TYPE ST_EtherCATSlaveInfo :
STRUCT
	nAddr 			: UDINT;
	nlinkState		: UDINT;
	edeviceState	: ST_EcSlaveState;
	sType 			: STRING[16];
	sName 			: STRING[32];
END_STRUCT
END_TYPE

(* stored: Version 1.1.0.1, ProductVersion 3.1.4024.15
   DUT ST_EtherCATSlaveInfo: Id {60ac04a1-ff09-493a-a681-f256502520e9} *)
